PROGRAM MAIN
VAR
    fbInfeed   : FB_Infeed;
    fbCapper   : FB_Capper;
    fbTransfer : FB_Transfer;
    fbScale    : FB_Scale;
    fbRecipe   : FB_RecipeHandler;
    fbLabeler  : FB_Labeler;
    nPerMinute : UDINT;
END_VAR

fbInfeed(bStart := GVL_Line.bAutoMode);
fbCapper(bStart := fbInfeed.bBottleInPlace);
fbTransfer(bRequest := fbCapper.bDone, fTarget := 250.0);
fbScale();
fbLabeler(nLabels := GVL_Line.nCapsDone);
nPerMinute := F_Throughput(nCaps := GVL_Line.nCapsDone,
                           nCycleTimeMs := GVL_Line.nCycleTimeMs);

END_PROGRAM

(* stored: Version 1.1.0.1, ProductVersion 3.1.4024.0
   POU MAIN: Id {d757552f-cf1f-43f5-9da6-13a3ce96c1a5}, SpecialFunc None *)
